Fanuc KAREL source: kb00128.KL

PROGRAM KB00128
%STACKSIZE=65535
%PRIORITY=65535
%NOLOCKGROUP
VAR
P1 : POSITION
-- UNRESOLVED DECLARATIONS (source type spelling not recovered)
-- RESULT : TYPE_0x0013 (type_u16=0x0013)
BEGIN
RESULT=ORIENT(P1)
END KB00128
